FUNCTION_BLOCK PML_StatePattern_Base
VAR_INPUT
END_VAR
VAR_OUTPUT
END_VAR
VAR
	stateMachine : PMLStateMachine;
	iStateMachine : IPmlStateMachine := stateMachine;
	undefined : Undefined_State(THIS, iStateMachine);
	aborting : Aborting_State(THIS, iStateMachine);
	aborted : Aborted_State(THIS, iStateMachine);
	clearing : Clearing_State(THIS, iStateMachine);
	stopped : Stopped_State(THIS, iStateMachine);
	resetting : Resetting_State(THIS, iStateMachine);
	idle : Idle_State(THIS, iStateMachine);
	starting : Starting_State(THIS, iStateMachine);
	execute : Execute_State(THIS, iStateMachine);
	iState : ITF_State := undefined;
END_VAR

iState.Cycle();
stateMachine();

METHOD SetState : BOOL
VAR_INPUT
  newState : ITF_State;
END_VAR
THIS^.iState := newState;
END_METHOD

END_FUNCTION_BLOCK

(* stored: Version 1.1.0.1, ProductVersion 3.1.4024.11
   POU PML_StatePattern_Base: Id {d1183f62-92d7-4751-9312-0004156ee9cc}, SpecialFunc None
   Method SetState: Id {2ca6654e-4c3f-4cc7-b3d6-deb3ce0ce962} *)
